# EPICS autosave request: iocBoot/iocARAmp/auto_settings_ARAmp75250AM2.req
file "aramp_settings_75250AM2.req",                P=$(P),  R=$(R)
